TYPE ST_APP_CTRL :
STRUCT
  Cmd       : E_INSTANCE_CMD;
  Variant   : E_APP_VARIANT;
END_STRUCT
END_TYPE

(* stored: Version 1.1.0.1, ProductVersion 3.1.4026.13
   DUT ST_APP_CTRL: Id {df31154c-b784-4bef-8cca-12faddca3455} *)
